{attribute 'GeneratedUsingTerminal: ER8309-1022-0018'}
{attribute addProperty BoxType "ER8309-1022-0018"}
{attribute addProperty Id "Enable_ditheringBOOL1EnableBOOL1ResetBOOL1"}
{attribute addProperty CRC "625230245"}
{attribute addProperty Size "3"}
TYPE Control_254441A5 :
STRUCT
	{attribute addProperty Name "Enable_dithering"}
	Enable_dithering : BOOL;
	{attribute addProperty Name "Enable"}
	Enable : BOOL;
	{attribute addProperty Name "Reset"}
	Reset : BOOL;
END_STRUCT
END_TYPE

(* stored: Version 1.2.0.0, ProductVersion 3.1.4024.9
   DUT Control_254441A5: Id {5c02e8bd-1169-4ba0-ba5c-fef6b0f4f596} *)
